TYPE ST_LaserGate :
STRUCT
	xIN	:	BOOL;
END_STRUCT
END_TYPE

(* stored: Version 1.1.0.1, ProductVersion 3.1.0.24
   DUT ST_LaserGate: Id {014fede3-11e7-4413-89b0-a3f559457f1b} *)
